(* CODESYS project Structure_RECOVERED_2024-06-28T13-38-27.project

Project tree, tasks and I/O mapping:
  Device : CODESYS Control Win V3, CODESYS, version 3.5.20.0
    application Application
      libraries: Standard, 3.5.18.0 (System)
      task MainTask (cyclic, interval t#20ms, priority 1) calls PLC_PRG
      program PLC_PRG [ST]
      data type myStruct
*)

// Device/Application/myStruct
TYPE myStruct :
STRUCT
	start:BOOL:=FALSE;
	
END_STRUCT
END_TYPE

// Device/Application/PLC_PRG
PROGRAM PLC_PRG
VAR
END_VAR

END_PROGRAM
